# B&R Automation Studio project POMiRTS-lab2
Automation Studio 4.5.2.102

## Configuration Config1

### Task classes (Cpu.sw)
```
Cyclic#1:
  ncsdcctrl <- ncsdcctrl.prg
Cyclic#4:
  Program <- Program.prg
NcDataObjects: acp10etxen <- acp10etxen.dob, gAxis01a <- gAxis01obj.gAxis01a.dob, gAxis01i <- gAxis01obj.gAxis01i.dob
Libraries: Acp10man, Acp10par, NcGlobal, Acp10sdc, Acp10_MC, brsystem, sys_lib, runtime, AsBrStr, DriveLib
```

### IoMap.iom - 4PP065_0571_P74/IoMap.iom
```iecst
VAR_CONFIG
	Cyclic#1.gAxis01_DrvIf.iLifeCnt AT %IB."8I64xxxxxxx.00x-1".SDC_LifeCnt;
	Cyclic#1.gAxis01_DrvIf.iDrvOK AT %IX."8I64xxxxxxx.00x-1".ETAD_Input_Bool_02;
	Cyclic#1.gAxis01_DrvIf.oSetTime AT %QW."8I64xxxxxxx.00x-1".SDC_SetTime;
	Cyclic#1.::stateMachine.speed AT %QW."8I64xxxxxxx.00x-1".LFRD_Output;
	Cyclic#1.gAxis01_DiDoIf.iLifeCntDriveReady AT %IB."8I64xxxxxxx.00x-1".SDC_LifeCnt;
	Cyclic#1.gAxis01_DiDoIf.iLifeCntDriveEnable AT %IB."8I64xxxxxxx.00x-1".SDC_LifeCnt;
	Cyclic#1.gAxis01_DiDoIf.oDriveEnable AT %QX."8I64xxxxxxx.00x-1".CMDD_Output_Bool_00;
	Cyclic#1.gAxis01_ModuleOk AT %QX."8I64xxxxxxx.00x-1".CMDD_Output_Bool_01;
	Cyclic#1.gAxis01_ModuleOk AT %QX."8I64xxxxxxx.00x-1".CMDD_Output_Bool_02;
	Cyclic#1.gAxis01_ModuleOk AT %IX."8I64xxxxxxx.00x-1".ModuleOk;
	Cyclic#1.gAxis01_DiDoIf.oDriveEnable AT %QX."8I64xxxxxxx.00x-1".CMDD_Output_Bool_03;
	Cyclic#1.gAxis01_DiDoIf.iDriveReady AT %IX."8I64xxxxxxx.00x-1".ETAD_Input_Bool_02;
	stateMachine.state AT %IW."8I64xxxxxxx.00x-1".ETAD_Input;
	stateMachine.command AT %QW."8I64xxxxxxx.00x-1".CMDD_Output;
	ledSM.led1 AT %QX."X20DO9322".DigitalOutput02;
	ledSM.led2 AT %QX."X20DO9322".DigitalOutput03;
	ledSM.led3 AT %QX."X20DO9322".DigitalOutput04;
	ledSM.led4 AT %QX."X20DO9322".DigitalOutput05;
	doorSM.direction AT %IX."X20DI9371".DigitalInput01;
	doorSM.sw1 AT %IX."X20DI9371".DigitalInput02;
	doorSM.sw2 AT %IX."X20DI9371".DigitalInput03;
	doorSM.sw3 AT %IX."X20DI9371".DigitalInput04;
	doorSM.sw4 AT %IX."X20DI9371".DigitalInput05;
END_VAR
```

## Logical view

Binary libraries used (declarations not repeated): operator, runtime, astime, AsIecCon, Acp10man, Acp10par, NcGlobal, Acp10sdc, Acp10_MC, brsystem, sys_lib, AsBrStr

### Global.var
```iecst
VAR
	gAxis01 : ACP10AXIS_typ;
	gAxis01_HW : SdcHwCfg_typ := (0);
	gAxis01_DrvIf : SdcDrvIf16_typ := (0);
	gAxis01_DiDoIf : SdcDiDoIf_typ := (0);
	gAxis01_ModuleOk : BOOL := 0;
	doorSM : DoorStateMachine;
	ledSM : LedStateMachine;
	stateMachine : DriveStateMachine;
END_VAR
```

### Library Logical/Libraries/DriveLib (ANSIC)

#### Types.typ
```iecst
TYPE
	state :
		(
		ST_DEC_NEG := 9,
		ST_DEC_POS := 8,
		ST_NEG := 7,
		ST_POS := 6,
		ST_ACC_NEG := 5,
		ST_ACC_POS := 4,
		ST_CLOSE := 3,
		ST_OPEN := 2,
		ST_UNKNOWN := 1,
		ST_INIT := 0
		);
END_TYPE
```

#### Constants.var
```iecst
VAR CONSTANT
	CMD_ENABLE : UINT := 15;
	CMD_SHUTDOWN : UINT := 6;
	CMD_SWITCH_ON : UINT := 7;
	STATE_DISABLED : UINT := 64;
	STATE_READY : UINT := 33;
	STATE_SWITCHED_ON : UINT := 35;
END_VAR
```

#### DriveLib.fun
```iecst
{REDUND_ERROR} FUNCTION_BLOCK LedStateMachine (*TODO: Add your comment here*) (*$GROUP=User,$CAT=User,$GROUPICON=User.png,$CATICON=User.png*)
	VAR_INPUT
		state : state := ST_INIT;
	END_VAR
	VAR_OUTPUT
		led1 : BOOL;
		led2 : BOOL;
		led3 : BOOL;
		led4 : BOOL;
		timer : INT;
	END_VAR
END_FUNCTION_BLOCK

{REDUND_ERROR} FUNCTION_BLOCK DriveStateMachine (*TODO: Add your comment here*) (*$GROUP=User,$CAT=User,$GROUPICON=User.png,$CATICON=User.png*)
	VAR_INPUT
		state : UINT;
		enable : BOOL;
	END_VAR
	VAR_OUTPUT
		command : UINT;
		speed : INT;
	END_VAR
END_FUNCTION_BLOCK

{REDUND_ERROR} FUNCTION_BLOCK DoorStateMachine (*TODO: Add your comment here*) (*$GROUP=User,$CAT=User,$GROUPICON=User.png,$CATICON=User.png*)
	VAR_OUTPUT
		state : state := ST_INIT;
	END_VAR
	VAR_INPUT
		sw1 : BOOL;
		sw2 : BOOL;
		sw3 : BOOL;
		sw4 : BOOL;
		direction : BOOL;
	END_VAR
	VAR_OUTPUT
		speed : INT;
	END_VAR
END_FUNCTION_BLOCK
```

#### DoorStateMachine.c
```c
#include <bur/plctypes.h>
#ifdef __cplusplus
	extern "C"
	{
#endif
#include "DriveLib.h"
#ifdef __cplusplus
	};
#endif
/* TODO: Add your comment here */
void DoorStateMachine(struct DoorStateMachine* inst)
{
	//
	switch (inst->state){
		/*
			Для согласованности индикации, тумблера, отвечающего за направление, и кнопок,
		отвечающих за датчики, направление ворот, в отличие от методички, выбрано так, что
		открытое состояние, когда ворота слева, и закрытое - справа. Т.о. direction == 0
		обозначает направление влево(открытие), а direction == 1 - вправо(закрытие)
		*/
		case ST_INIT:
			inst->speed = 0;
			inst->state=ST_UNKNOWN;
			break;

		case ST_UNKNOWN:
			/*
				Из неизвестного состяния мы можем перейти в одно из двух, открыты или закрыты.
			При этом помимо направления, также должен быть задействован соответствующий датчик,
			иначе остаемся в неизвестном состоянии
			*/
			if (inst->sw1 && inst->direction == 0){
				inst->state = ST_OPEN;
				break;
			} else if (inst->sw4 && inst->direction == 1){
				inst->state = ST_CLOSE;
				break;
			} else {
				inst->speed = (inst->direction == 0)?-50:50;
				break;
			}

		case ST_OPEN:
			/*
				Если ворота открыты, а направление остаётся тем же (влево), то скорость остаётся нулевой, остаёмся в том же состоянии.
			Иначе, если направление теперь другое (вправо) то переход в состояние ACC_POS (узкорение в сторону закрытия (вправо).
			В случае неизвестной комбинации сигналов с датчиков - отправка в состояние UNKNOWN.
			*/
			// Остаемся в ST_OPEN
			if (inst->direction == 0){
				inst->speed = 0;
				break;
			}
			// Переход в ST_ACC_POS
			else if (inst->direction == 1){
				inst->state = ST_ACC_POS;
				break;
			}
			// Переход в UNKNOWN
			else {
				inst->state = ST_UNKNOWN;
				break;
			}

		case ST_ACC_POS:
			/*
				Если ворота ускоряются, то они остюаются в том же положении пока не сработал второй датчик
			или не изменилось направление. Когда сработал второй датчик, то устанавливается максимальная
			скорость и состояние ST_POS. Когда меняется направление, то устанавливается обратная скорость
			и состояние ST_DEC_NEG
			*/
			// Остаемся в ST_ACC_POS
			if (inst->direction == 1 && !inst->sw2){
				inst->speed = 100;
				break;
			}
			// Сработал второй датчик, переход в ST_POS
			else if (inst->direction == 1 && inst->sw2){
				inst->state = ST_POS;
				break;
			}
			// Изменилось направление, переход в ST_DEC_NEG, установка обратной скорости
			else if (inst->direction == 0) {
				inst->state = ST_DEC_NEG;
				break;
			}
			// Неизвестное состояние
			else {
				inst->speed = 0;
				inst->state = ST_UNKNOWN;
				break;
			}

		case ST_POS:
			/*
				Состояние максимальной скорости, движение в сторону закрытия. Остаёмся в том же состоянии пока не сработал третий датчик.
			После срабатывания третьего датчика переход в ST_DEC_POS. Если сменится направление то переход в ST_NEG.
			*/
			// То же состояние
			if (inst->direction == 1 && !inst->sw3){
				inst->speed = 200;
				break;
			}
			// Сработал 3 датчик, замедление
			else if (inst->direction == 1){
				inst->state = ST_DEC_POS;
				break;
			}
			// Смена направления
			else if (inst->direction == 0){
				inst->state = ST_NEG;
				break;
			}
			// Неизвестное состояние
			else{
				inst->state = ST_UNKNOWN;
				break;
			}

		case ST_DEC_POS:
			/*
				Состояние замедления перед закрытием. При отстутсвии новых сигналов остаётся в том же состоянии. При наличии сигнала с последнего
			датчика переход в состояние ST_CLOSE. При смене направления, переход в состояние ST_ACC_NEG. Иначе ST_UNKNOWN.
			*/
			// Сохранение состояния
			if (inst->direction == 1 && !inst->sw4){
				inst->speed=100;
				break;
			}
			// Переход в закрытое состояние
			else if (inst->direction == 1 && inst->sw4)
			{
				inst->state = ST_CLOSE;
				break;
			}
			// Смена направления
			else if (inst->direction == 0)
			{
				inst->state = ST_ACC_NEG;
				break;
			}
			// Переход в неизвестное состояние
			else{
				inst->state = ST_UNKNOWN;
				break;
			}

		case ST_CLOSE:
			if (inst->direction == 1)
			{
				inst->speed = 0;
				break;
			}
			else if(inst->direction == 0){
				inst->state = ST_ACC_NEG;
				break;
			}
			else
			{
				inst->state = ST_UNKNOWN;
				break;
			}

		case ST_ACC_NEG:
			/*
				Состояние открывающихся ворот, сохраняет состояние пока не сработает 3 датчик или не изменится направление
			*/
			if (inst->direction == 0 && !inst->sw3){
				inst->speed = -100;
				break;
			}
			else if (inst->sw3){
				inst->state = ST_NEG;
				break;
			}
			else if (inst->direction == 1){
				inst->state = ST_DEC_POS;
				break;
			}
			else {
				inst->state = ST_UNKNOWN;
				break;
			}

		case ST_NEG:
			/*Открытие ворот на макс скорости*/
			if (inst->direction == 0 && !inst->sw2){
				inst->speed = -200;
				break;
			}
			else if (inst->direction == 0) {
				inst->state = ST_DEC_NEG;
				break;
			}
			else if (inst->direction == 1){
				inst->state = ST_POS;
				break;
			}
			else{
				inst->state = ST_UNKNOWN;
				break;
			}
		case ST_DEC_NEG:
			if (inst->direction == 0 && !inst->sw1){
				inst->speed = -100;
				break;
			}
			else if(inst->direction == 0){
				inst->state = ST_OPEN;
				break;
			}
			else if (inst->direction == 1){
				inst->state = ST_ACC_POS;
				break;
			}
			else {
				inst->state = ST_UNKNOWN;
				break;
			}

	}
}
```

#### DriveStateMachine.c
```c
#include <bur/plctypes.h>
#ifdef __cplusplus
	extern "C"
	{
#endif
	#include "DriveLib.h"
#ifdef __cplusplus
	};
#endif
/* TODO: Add your comment here */
void DriveStateMachine(struct DriveStateMachine* inst)
{
	/*TODO: Add your code here*/
	UINT mask = inst->state & 0x6f;
	if(!inst->enable){
		inst->command = CMD_SHUTDOWN;
	}
	else{
		switch (mask){
			case STATE_DISABLED:
				inst->command = CMD_SHUTDOWN;
				break;

			case STATE_READY:
				inst->command = CMD_ENABLE;
				break;

			case STATE_SWITCHED_ON:
				inst->command = CMD_SWITCH_ON;
				break;
		}
	}
}
```

#### LedStateMachine.c
```c
#include <bur/plctypes.h>
#ifdef __cplusplus
	extern "C"
	{
#endif
	#include "DriveLib.h"
#ifdef __cplusplus
	};
#endif
/* TODO: Add your comment here */
void LedStateMachine(struct LedStateMachine* inst)
{
	switch(inst->state){
		case ST_INIT:
			inst->led1 = 0;
			inst->led2 = 0;
			inst->led3 = 0;
			inst->led4 = 0;
			break;

		case ST_UNKNOWN:
			if (inst->timer%10==0){
				inst->led1=!inst->led1;
				inst->led2=!inst->led2;
				inst->led3=!inst->led3;
				inst->led4=!inst->led4;
			}
			break;

		case ST_OPEN:
			inst->led1 = 0;
			inst->led2 = 0;
			inst->led3 = 0;
			inst->led4 = 0;
			break;

		case ST_ACC_POS:
			inst->led1 = 1;
			inst->led2 = 0;
			inst->led3 = 0;
			inst->led4 = 0;
			break;

		case ST_POS:
			inst->led1 = 1;
			inst->led2 = 1;
			inst->led3 = 0;
			inst->led4 = 0;
			break;

		case ST_DEC_POS:
			inst->led1 = 1;
			inst->led2 = 1;
			inst->led3 = 1;
			inst->led4 = 0;
			break;

		case ST_CLOSE:
			inst->led1 = 1;
			inst->led2 = 1;
			inst->led3 = 1;
			inst->led4 = 1;
			break;

		case ST_ACC_NEG:
			inst->led1 = 1;
			inst->led2 = 1;
			inst->led3 = 1;
			inst->led4 = 0;
			break;

		case ST_NEG:
			inst->led1 = 1;
			inst->led2 = 1;
			inst->led3 = 0;
			inst->led4 = 0;
			break;

		case ST_DEC_NEG:
			inst->led1 = 1;
			inst->led2 = 0;
			inst->led3 = 0;
			inst->led4 = 0;
			break;
	}
}
```

### Program Logical/Program

#### Variables.var
```iecst
VAR
	timeCounter : USINT := 0;
END_VAR
```

#### Main.c
```c
#include <bur/plctypes.h>

#ifdef _DEFAULT_INCLUDES
	#include <AsDefault.h>
#endif

void _INIT ProgramInit(void)
{
	stateMachine.enable = 1;
}

void _CYCLIC ProgramCyclic(void)
{
	timeCounter++;
	ledSM.timer = timeCounter;
	ledSM.state = doorSM.state;
	DoorStateMachine(&doorSM);
	LedStateMachine(&ledSM);
	stateMachine.speed = doorSM.speed;
	DriveStateMachine(&stateMachine);
}

void _EXIT ProgramExit(void)
{

}
```
